PROGRAM Laser_Marking
VAR
END_VAR

END_PROGRAM

(* stored: Version 1.1.0.1, ProductVersion 3.1.4024.11
   POU Laser_Marking: Id {8db33281-600b-47e0-abaa-d1b44fe04a7e}, SpecialFunc None *)
